Staubli VAL3: sockets.dtx

public sio skCognex[10]
  [0] = {link=Socket\cognex1}
  [1] = {link=Socket\cognex2}
  [2] = {link=Socket\cognex3}
  [3] = {link=Socket\cognex4}
  [4] = {link=Socket\cognex5}
  [5] = {link=Socket\cognex6}
  [6] = {link=Socket\cognex7}
  [7] = {link=Socket\cognex8}
  [8] = {link=Socket\cognex9}
  [9] = {link=Socket\cognex10}
public sio skFromRobot[10]
  [0] = {link=Socket\fromRobot_sk1}
  [1] = {link=Socket\fromRobot_sk2}
  [2] = {link=Socket\fromRobot_sk3}
  [3] = {link=Socket\fromRobot_sk4}
  [4] = {link=Socket\fromRobot_sk5}
  [5] = {link=Socket\fromRobot_sk6}
  [6] = {link=Socket\fromRobot_sk7}
  [7] = {link=Socket\fromRobot_sk8}
  [8] = {link=Socket\fromRobot_sk9}
  [9] = {link=Socket\fromRobot_sk10}
